TYPE DataTag :
STRUCT
	{attribute 'TagName' := 'machine_id'}
    machine_id : STRING;
	{attribute 'TagName' := 'module_name'}
    module_name: STRING;
END_STRUCT
END_TYPE

(* stored: Version 1.1.0.1, ProductVersion 3.1.4024.12
   DUT DataTag: Id {0ab55ead-4543-4a85-afed-636ac6c930a0} *)
